// Mitsubishi GX Works2 project: SmartFarmDXz   PLC: FX3U/FX3UC

PROGRAM MAIN
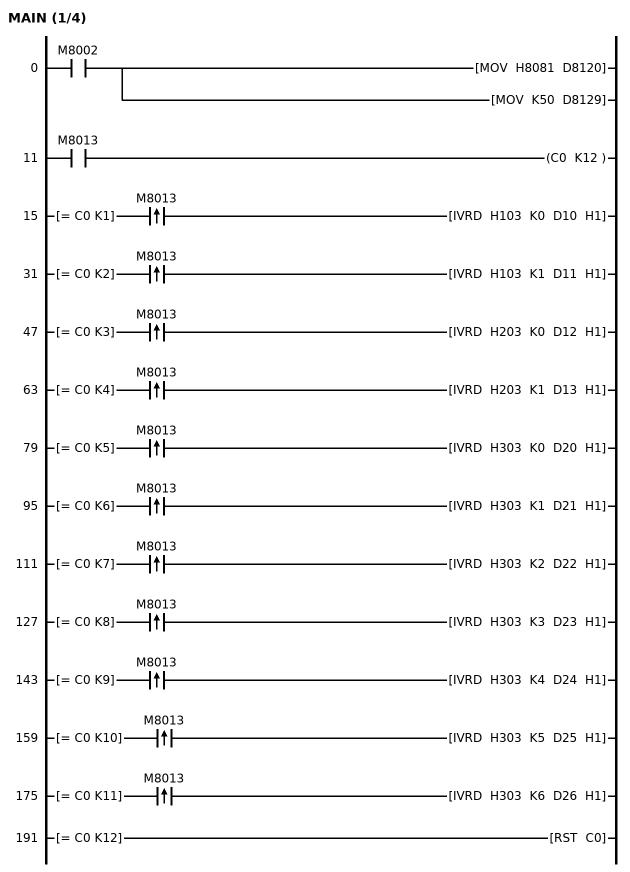
0     LD      M8002
      MOV     H8081 D8120
      MOV     K50 D8129
11    LD      M8013
      OUT     C0 K12
15    LD=     C0 K1
      ANDP    M8013
      IVRD    H103 K0 D10 H1
31    LD=     C0 K2
      ANDP    M8013
      IVRD    H103 K1 D11 H1
47    LD=     C0 K3
      ANDP    M8013
      IVRD    H203 K0 D12 H1
63    LD=     C0 K4
      ANDP    M8013
      IVRD    H203 K1 D13 H1
79    LD=     C0 K5
      ANDP    M8013
      IVRD    H303 K0 D20 H1
95    LD=     C0 K6
      ANDP    M8013
      IVRD    H303 K1 D21 H1
111   LD=     C0 K7
      ANDP    M8013
      IVRD    H303 K2 D22 H1
127   LD=     C0 K8
      ANDP    M8013
      IVRD    H303 K3 D23 H1
143   LD=     C0 K9
      ANDP    M8013
      IVRD    H303 K4 D24 H1
159   LD=     C0 K10
      ANDP    M8013
      IVRD    H303 K5 D25 H1
175   LD=     C0 K11
      ANDP    M8013
      IVRD    H303 K6 D26 H1
191   LD=     C0 K12
      RST     C0
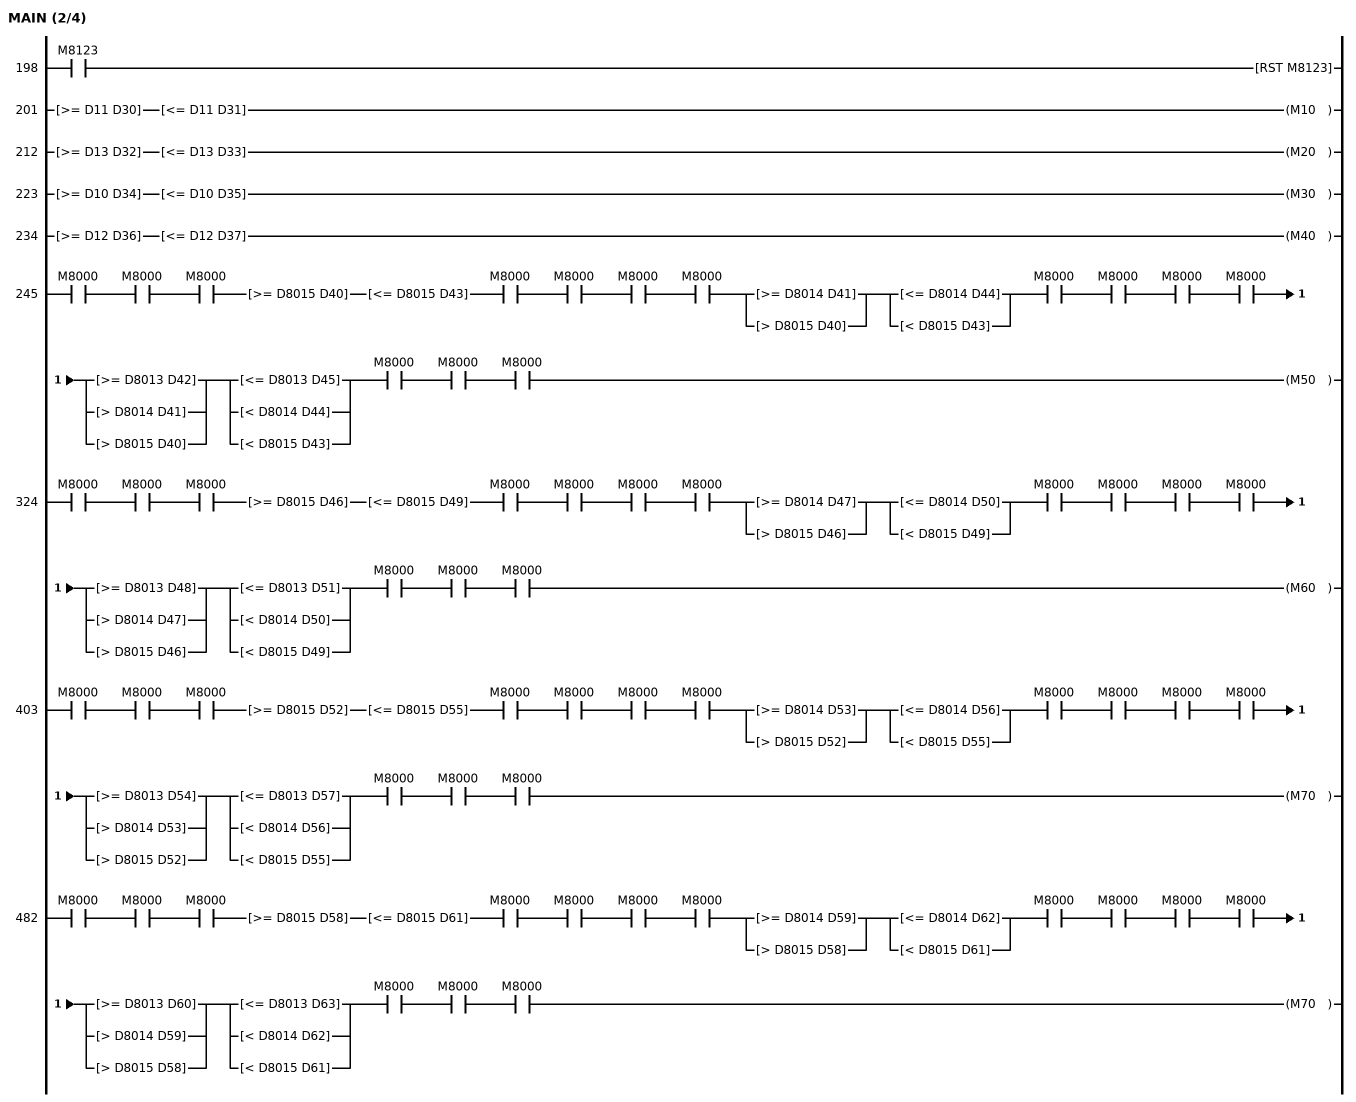
198   LD      M8123
      RST     M8123
201   LD>=    D11 D30
      AND<=   D11 D31
      OUT     M10
212   LD>=    D13 D32
      AND<=   D13 D33
      OUT     M20
223   LD>=    D10 D34
      AND<=   D10 D35
      OUT     M30
234   LD>=    D12 D36
      AND<=   D12 D37
      OUT     M40
245   LD      M8000
      AND     M8000
      AND     M8000
      AND>=   D8015 D40
      AND<=   D8015 D43
      AND     M8000
      AND     M8000
      AND     M8000
      AND     M8000
      LD>=    D8014 D41
      OR>     D8015 D40
      ANB
      LD<=    D8014 D44
      OR<     D8015 D43
      ANB
      AND     M8000
      AND     M8000
      AND     M8000
      AND     M8000
      LD>=    D8013 D42
      OR>     D8014 D41
      OR>     D8015 D40
      ANB
      LD<=    D8013 D45
      OR<     D8014 D44
      OR<     D8015 D43
      ANB
      AND     M8000
      AND     M8000
      AND     M8000
      OUT     M50
324   LD      M8000
      AND     M8000
      AND     M8000
      AND>=   D8015 D46
      AND<=   D8015 D49
      AND     M8000
      AND     M8000
      AND     M8000
      AND     M8000
      LD>=    D8014 D47
      OR>     D8015 D46
      ANB
      LD<=    D8014 D50
      OR<     D8015 D49
      ANB
      AND     M8000
      AND     M8000
      AND     M8000
      AND     M8000
      LD>=    D8013 D48
      OR>     D8014 D47
      OR>     D8015 D46
      ANB
      LD<=    D8013 D51
      OR<     D8014 D50
      OR<     D8015 D49
      ANB
      AND     M8000
      AND     M8000
      AND     M8000
      OUT     M60
403   LD      M8000
      AND     M8000
      AND     M8000
      AND>=   D8015 D52
      AND<=   D8015 D55
      AND     M8000
      AND     M8000
      AND     M8000
      AND     M8000
      LD>=    D8014 D53
      OR>     D8015 D52
      ANB
      LD<=    D8014 D56
      OR<     D8015 D55
      ANB
      AND     M8000
      AND     M8000
      AND     M8000
      AND     M8000
      LD>=    D8013 D54
      OR>     D8014 D53
      OR>     D8015 D52
      ANB
      LD<=    D8013 D57
      OR<     D8014 D56
      OR<     D8015 D55
      ANB
      AND     M8000
      AND     M8000
      AND     M8000
      OUT     M70
482   LD      M8000
      AND     M8000
      AND     M8000
      AND>=   D8015 D58
      AND<=   D8015 D61
      AND     M8000
      AND     M8000
      AND     M8000
      AND     M8000
      LD>=    D8014 D59
      OR>     D8015 D58
      ANB
      LD<=    D8014 D62
      OR<     D8015 D61
      ANB
      AND     M8000
      AND     M8000
      AND     M8000
      AND     M8000
      LD>=    D8013 D60
      OR>     D8014 D59
      OR>     D8015 D58
      ANB
      LD<=    D8013 D63
      OR<     D8014 D62
      OR<     D8015 D61
      ANB
      AND     M8000
      AND     M8000
      AND     M8000
      OUT     M70
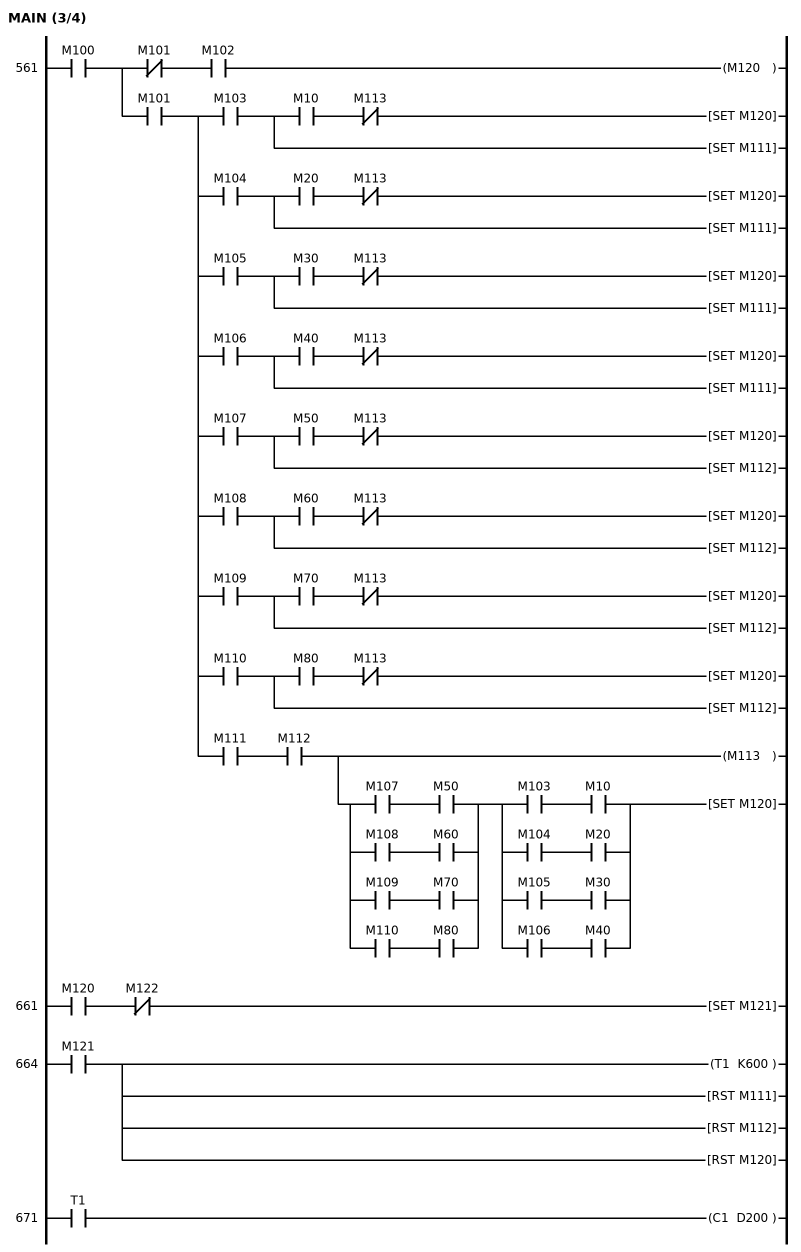
561   LD      M100
      MPS
      ANI     M101
      AND     M102
      OUT     M120
      MPP
      AND     M101
      MPS
      AND     M103
      MPS
      AND     M10
      ANI     M113
      SET     M120
      MPP
      SET     M111
      MRD
      AND     M104
      MPS
      AND     M20
      ANI     M113
      SET     M120
      MPP
      SET     M111
      MRD
      AND     M105
      MPS
      AND     M30
      ANI     M113
      SET     M120
      MPP
      SET     M111
      MRD
      AND     M106
      MPS
      AND     M40
      ANI     M113
      SET     M120
      MPP
      SET     M111
      MRD
      AND     M107
      MPS
      AND     M50
      ANI     M113
      SET     M120
      MPP
      SET     M112
      MRD
      AND     M108
      MPS
      AND     M60
      ANI     M113
      SET     M120
      MPP
      SET     M112
      MRD
      AND     M109
      MPS
      AND     M70
      ANI     M113
      SET     M120
      MPP
      SET     M112
      MRD
      AND     M110
      MPS
      AND     M80
      ANI     M113
      SET     M120
      MPP
      SET     M112
      MPP
      AND     M111
      AND     M112
      OUT     M113
      LD      M107
      AND     M50
      LD      M108
      AND     M60
      ORB
      LD      M109
      AND     M70
      ORB
      LD      M110
      AND     M80
      ORB
      ANB
      LD      M103
      AND     M10
      LD      M104
      AND     M20
      ORB
      LD      M105
      AND     M30
      ORB
      LD      M106
      AND     M40
      ORB
      ANB
      SET     M120
661   LD      M120
      ANI     M122
      SET     M121
664   LD      M121
      OUT     T1 K600
      RST     M111
      RST     M112
      RST     M120
671   LD      T1
      OUT     C1 D200
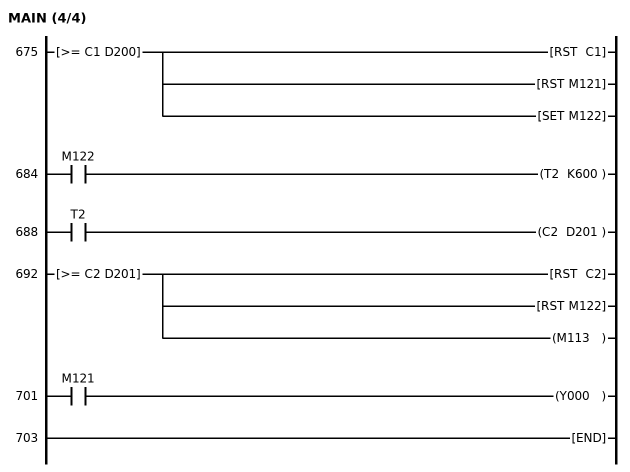
675   LD>=    C1 D200
      RST     C1
      RST     M121
      SET     M122
684   LD      M122
      OUT     T2 K600
688   LD      T2
      OUT     C2 D201
692   LD>=    C2 D201
      RST     C2
      RST     M122
      OUT     M113
701   LD      M121
      OUT     Y000
703   END
END_PROGRAM
